// ════════════════════════════════════════════════════════════════
// 3. APLICA OFFSET AO TIMESTAMP UTC
// ════════════════════════════════════════════════════════════════

// ✅ MÉTODO SEGURO: Usa valor absoluto e subtrai/soma conforme sinal
offsetSeconds_ABS := DINT_TO_UDINT(ABS(offsetSeconds));

IF offsetSeconds < 0 THEN
    // Fuso NEGATIVO (Américas): subtrai
    timestampLocal_UDINT := Global.timestampUTC - offsetSeconds_ABS;
ELSE
    // Fuso POSITIVO (Europa, Ásia): soma
    timestampLocal_UDINT := Global.timestampUTC + offsetSeconds_ABS;
END_IF

// ════════════════════════════════════════════════════════════════
// 4. CONVERTE TIMESTAMP PARA DATA/HORA LOCAL
// ════════════════════════════════════════════════════════════════

dtNowLocal := UDINT_TO_DT(timestampLocal_UDINT);
dataNowLocal := TO_DATE(dtNowLocal);

// Extrai hora (0..23)
todNowLocal := DT_TO_TOD(dtNowLocal);
todAsDword := TOD_TO_DWORD(todNowLocal);
hora := DWORD_TO_INT(todAsDword / DWORD#3600000);

// Extrai dia da semana (1=Dom .. 7=Sáb)
diadasemana := UDINT_TO_INT(((timestampLocal_UDINT / 86400) + 4) MOD 7) + 1;

// ════════════════════════════���═══════════════════════════════════
// 5. VERIFICA MUDANÇA DE DATA (Para atualizar cache)
// ════════════════════════════════════════════════════════════════

IF dataNowLocal <> lastCheckedDate THEN
    
    lastCheckedDate := dataNowLocal;
    cachedSpecialDateLimit := -1.0;  // Invalida cache
    
    FOR i := 1 TO Global.NDATASESPECIAIS DO
        
        // ✅ OTIMIZAÇÃO: Early exit se encontrar data vazia
        IF PerVar.DatasEspeciais[i] = DATE#1970-01-01 THEN
            EXIT;  // Resto do array está vazio
        END_IF
        
        // Verifica se é data especial
        IF PerVar.DatasEspeciais[i] = dataNowLocal THEN
            cachedSpecialDateLimit := PerVar.SpecialDaySchedule[i];
            EXIT;  // Encontrou, pára a busca
        END_IF
        
    END_FOR
    
END_IF

// ════════════════════════════════════════════════════════════════
// 6. USA CACHE DE DATA ESPECIAL (Se válido)
// ════════════════════════════════════════════════════════════════

IF cachedSpecialDateLimit >= 0.0 THEN
    // Data especial ativa
    Global.MaxExportLimit := cachedSpecialDateLimit;
    Global.sMessage := 'Agenda: Data especial';
    RETURN;
END_IF

// ════════════════════════════════════════════════════════════════
// 7. AGENDA SEMANAL (Hora Local)
// ════════════════════════════════════════════════════════════════

// ✅ VALIDAÇÃO: Verifica se índices estão dentro dos limites
IF (diadasemana >= 1 AND diadasemana <= 7) AND (hora >= 0 AND hora <= 23) THEN
    
    // Acessa agenda semanal
    Global.MaxExportLimit := PerVar.WeekSchedule_kW[diadasemana, hora + 1];
    Global.sMessage := '';  // ✅ Limpa mensagem de erro anterior
    
ELSE
    
    // ❌ ERRO: Índice inválido (não deveria ocorrer)
    Global.MaxExportLimit := 0.0;
    Global.sMessage := 'ERRO: Índice de agenda inválido';
    Global.K8ErroOut := TRUE;
    
END_IF

END_FUNCTION_BLOCK

// Dispositivo/Application/FB Auxiliares/FB_FFQ
(*
    FB_FFQ - Feedforward de Potência Reativa 
    Função:
    - Calcula o Q MÍNIMO necessário para atingir PF_target
    - Não calcula Q exato, mas o valor mínimo aceitável
    - Se o sistema fornecer menos Q, o PF ficará maior (melhor)
    - Se fornecer mais Q, o PF ficará menor (pior)
    Fórmula:
    Q_min = P × tan(acos(PF_target)) => Simplificado: Q_min = P × √(1 - PF²) / PF
*)

FUNCTION_BLOCK FB_FFQ
VAR_INPUT
    P_active_kW   : REAL;    // Potência ativa comandada (kW)
    PF_target_abs : REAL;    // PF alvo (0.92)
    PF_sign       : REAL;    // 1.0 = indutivo, -1.0 = capacitivo
END_VAR

VAR_OUTPUT
    Q_reactive_kvar : REAL;   // Potência Reativa Calculada (var) - Q mínimo para atingir PF_target
END_VAR

VAR
    tan_phi : REAL;           // Tangente do ângulo de fase
    Q_target    : REAL;       // Q total necessário no ponto de conexão
END_VAR

// 1. Proteção: se potência ativa é zero ou negativa, não há Q a calcular
IF P_active_kW <= 0.0 THEN
    Q_reactive_kvar := 0.0;
    RETURN;
END_IF

// Proteção: PF_target deve estar entre 0 e 1
IF PF_target_abs <= 0.0 OR PF_target_abs > 1.0 THEN
    Q_reactive_kvar := 0.0;
    RETURN;
END_IF

// 2. Q total necessário no ponto de conexão para PF = 0.92
// Método 1: usando tan(acos(PF))
// phi := ACOS(PF_target_abs);              // Ângulo de fase em radianos
// tan_phi := TAN(phi);                     // Tangente do ângulo
// Q_reactive_var := P_active_W * tan_phi;
// Método 2: Simplificado (mais eficiente, evita ACOS e TAN)
// tan(acos(x)) = sqrt(1 - x²) / x
tan_phi := SQRT(1.0 - (PF_target_abs * PF_target_abs)) / PF_target_abs;
Q_target := P_active_kW * tan_phi;

// atribuição correta
Q_reactive_kvar := Q_target;

// 3. Aplica o sinal (Indutivo = positivo, Capacitivo = negativo)
// Nota: Para controle de exportação, normalmente usamos indutivo (Q positivo)
IF PF_sign < 0.0 THEN
    Q_reactive_kvar := -Q_reactive_kvar;  // Capacitivo
END_IF

// Resultado: Q_reactive_var é o Q MÍNIMO para atingir PF_target
// - Se injetar menos Q: PF > PF_target (melhor)
// - Se injetar mais Q: PF < PF_target (pior)
// - Se injetar exatamente Q: PF = PF_target

END_FUNCTION_BLOCK

// Dispositivo/Application/FB Auxiliares/FB_PIQ
(*
    FB_PIQ - Controlador PI para Fator de Potência
    Lógica para PF ≥ 0.92:
    - Se PV (PF medido) ≥ SP (PF target): erro = 0 (objetivo atingido)
    - Se PV < SP: erro = SP - PV (precisa aumentar Q)
    Diferente de um PI normal:
    - Erro ZERO quando PF ≥ target (não tenta melhorar além do necessário)
    - Saída é comando de Q (kvar)
*)

FUNCTION_BLOCK FB_PIQ
VAR_INPUT
    SP : REAL;                      		// Setpoint de PF (0.92)
    PV : REAL;                      		// PF medido (absoluto)
	Kp : REAL;              
    Ki : REAL;              
    CycleTime : REAL;       				
    P_cmd : REAL;                   		// Comando de P (para referência)
    RampUp : REAL;                  		// Rampa de subida (kvar/s)
    RampDown : REAL;                		// Rampa de descida (kvar/s)
    DeadbandAbs : REAL;             		// Zona morta de PF (ex: 0.01)
    Reset : BOOL;                   		// Zera o controlador
    bExternal_Saturated : BOOL := FALSE;  	// NOVO: Saturação externa (de FB_QAlloc)
	OutMax : REAL := 1000.0;    			// Limite superior de MV (kvar)
    OutMin : REAL := 0.0;       			// Limite inferior de MV (kvar)
END_VAR

VAR_OUTPUT
    MV : REAL;                      // Comando de Q (kvar)
    Error : REAL;                   // BOOL → REAL (valor do erro)
    Saturated : BOOL;               // TRUE = saída saturada
END_VAR

VAR
    integral : REAL := 0.0;         // Acumulador integral
    P_term : REAL;                  // Termo proporcional
    I_term : REAL;                  // Termo integral
    MV_raw : REAL;                  // Saída bruta (antes de rampa)
    MV_prev : REAL := 0.0;          // Saída do ciclo anterior
    delta : REAL;                   // Variação desejada
    delta_max : REAL;               // Variação máxima permitida
    erro : REAL;                    // Erro de PF
    sinal_saturacao : INT;      	// para anti-windup direcional
END_VAR

// ════════════════════════════════════════════════════════════════
// 1. RESET
// ════════════════════════════════════════════════════════════════
IF Reset THEN
    integral := 0.0;
    MV := 0.0;
    MV_prev := 0.0;
    Error := 0.0;  
    Saturated := FALSE;
    RETURN;
END_IF

// ════════════════════════════════════════════════════════════════
// 2. CALCULA ERRO COM LÓGICA ESPECIAL (PF ≥ TARGET)
// ════════════════════════════════════════════════════════════════

IF PV >= SP THEN
    erro := 0.0;  // PF medido ≥ PF target: objetivo atingido
ELSE
    erro := SP - PV;  // PF medido < PF target: precisa corrigir
END_IF

Error := erro;  // ✅ Saída do erro

// ════════════════════════════════════════════════════════════════
// 3. ZONA MORTA (DEADBAND)
// ════════════════════════════════════════════════════════════════

IF ABS(erro) < DeadbandAbs THEN
    erro := 0.0;
END_IF

// ════════════════════════════════════════════════════════════════
// 4. CÁLCULO PI
// ════════════════════════════════════════════════════════════════

P_term := Kp * erro;
I_term := integral + (Ki * erro * CycleTime);
MV_raw := P_term + I_term;

// ════════════════════════════════════════════════════════════════
// 5. ✅ SATURAÇÃO COM OutMax/OutMin (ALTERAÇÃO)
// ════════════════════════════════════════════════════════════════
IF MV_raw > OutMax THEN
    MV_raw := OutMax;
    sinal_saturacao := 1;
ELSIF MV_raw < OutMin THEN
    MV_raw := OutMin;
    sinal_saturacao := -1;
ELSE
    sinal_saturacao := 0;
END_IF

// ════════════════════════════════════════════════════════════════
// 6. ANTI-WINDUP (Conditional Integration)
// ════════════════════════════════════════════════════════════════

IF bExternal_Saturated OR (sinal_saturacao <> 0) THEN
    // Saturado: só acumula se erro empurra para FORA da saturação
    IF (sinal_saturacao = 1 AND erro < 0.0) OR
       (sinal_saturacao = -1 AND erro > 0.0) THEN
        integral := I_term;  // Permite desacumular
    END_IF
    // Caso contrário: integral permanece (freeze)
    Saturated := TRUE;
ELSE
    integral := I_term;
    Saturated := FALSE;
END_IF

// ════════════════════════════════════════════════════════════════
// 7. RATE LIMITER (Rampa)
// ════════════════════════════════════════════════════════════════

delta := MV_raw - MV_prev;

IF delta > 0.0 THEN
    delta_max := RampUp * Global.ControlCycle;
    IF delta > delta_max THEN
        MV := MV_prev + delta_max;
    ELSE
        MV := MV_raw;
    END_IF
    
ELSIF delta < 0.0 THEN
    delta_max := RampDown * Global.ControlCycle;
    IF ABS(delta) > delta_max THEN
        MV := MV_prev - delta_max;
    ELSE
        MV := MV_raw;
    END_IF
    
ELSE
    MV := MV_raw;
END_IF

MV_prev := MV;

END_FUNCTION_BLOCK

// Dispositivo/Application/FB Auxiliares/FB_QAlloc

(*
    ════════════════════════════════════════════════════════════════
    FB_QAlloc - Alocador de Potência Reativa
    ════════════════════════════════════════════════════════════════
*)

FUNCTION_BLOCK FB_QAlloc
VAR_INPUT
    Q_total_cmd_kvar : REAL;        // Comando de Q total (do FB_PIQ)
END_VAR

VAR_OUTPUT
    bQ_limit_reached : BOOL;        // TRUE = Não conseguiu alocar todo Q
    Q_allocated_kvar : REAL;        // Q efetivamente alocado
    PF_effective : REAL;            // PF efetivo total resultante
    Q_capacity_total : REAL;        // Capacidade total de Q disponível (kvar)
    S_total_used : REAL;            // S total utilizado (kVA)
END_VAR

VAR

	// ✅ Acumuladores totais
    Q_total : REAL;
    P_total : REAL;
    Q_capacity_total_internal : REAL;
    S_total_used_internal : REAL;

	// ✅ Variáveis por inversor
    Q_target_i : REAL;
    Q_actual_i : REAL;
    Q_max_i : REAL;
    S_available_i : REAL;
    P_actual_i : REAL;
	
    // ✅ Auxiliares
    i : UINT;
    proportion : REAL;
    S_total : REAL;
    S_i : REAL;  // ✅ S do inversor i (calculado 1 vez)
END_VAR

// ════════════════════════════════════════════════════════════════
// INICIALIZAÇÃO
// ════════════════════════════════════════════════════════════════

Q_total := 0.0;
P_total := 0.0;
Q_capacity_total_internal := 0.0;
S_total_used_internal := 0.0;
bQ_limit_reached := FALSE;

// ════════════════════════════════════════════════════════════════
// LOOP PRINCIPAL
// ════════════════════════════════════════════════════════════════

FOR i := 1 TO Global.NMAXINVERSORES DO
    
    IF PerVar.InvActivePower[i] > 0.0 THEN
        
        // ────────────────────────────────────────────────────────
        // A. LÊ P JÁ ALOCADO
        // ────────────────────────────────────────────────────────
        P_actual_i := Global.P_inv_kW[i];
        
        // ────────────────────────────────────────────────────────
        // B. CALCULA Q MÁXIMO DISPONÍVEL
        // ────────────────────────────────────────────────────────
        S_available_i := PerVar.InvSmaxPower[i];
        
        IF S_available_i > ABS(P_actual_i) THEN
            Q_max_i := SQRT((S_available_i * S_available_i) - (P_actual_i * P_actual_i));
        ELSE
            Q_max_i := 0.0;
        END_IF
        
        Global.Inv_Q_available[i] := Q_max_i;
        
        // ─────────────────────────────────────────���──────────────
        // C. DISTRIBUI Q PROPORCIONALMENTE
        // ────────────────────────────────────────────────────────
        IF Global.P_allocated_kW > 0.01 THEN
            proportion := Global.P_inv_kW[i] / Global.P_allocated_kW;
        ELSE
            proportion := 0.0;
        END_IF
        
        Q_target_i := Q_total_cmd_kvar * proportion;
        
        // ────────────────────────────────────────────────────────
        // D. LIMITA Q AO DISPONÍVEL
        // ────────────────────────────────────────────────────────
        IF ABS(Q_target_i) > Q_max_i THEN
            
            IF Q_target_i >= 0.0 THEN
                Q_actual_i := Q_max_i;
            ELSE
                Q_actual_i := -Q_max_i;
            END_IF
            
            bQ_limit_reached := TRUE;
            Global.Inv_limited[i] := TRUE;
            
        ELSE
            Q_actual_i := Q_target_i;
            Global.Inv_limited[i] := FALSE;
        END_IF
        
        // ────────────────────────────────────────────────────────
        // E. ARMAZENA Q
        // ────────────────────���───────────────────────────────────
        Global.Q_inv_kvar[i] := Q_actual_i;
        
        // ────────────────────────────────────────────────────────
        // F. CALCULA S UTILIZADO (✅ UMA VEZ)
        // ────────────────────────────────────────────────────────
        S_i := SQRT((P_actual_i * P_actual_i) + (Q_actual_i * Q_actual_i));
        
        S_total_used_internal := S_total_used_internal + S_i;
        
        // Utilização de S (%)
        IF S_available_i > 0.0 THEN
            Global.Inv_S_utilization[i] := (S_i / S_available_i) * 100.0;
        ELSE
            Global.Inv_S_utilization[i] := 0.0;
        END_IF
        
        // ────────────────────────────────────────────────────────
        // G. CALCULA PF INDIVIDUAL
        // ────────────────────────────────────────────────────────
        IF S_i > 0.01 THEN
            Global.PF_inv[i] := P_actual_i / S_i;
        ELSE
            Global.PF_inv[i] := 1.0;
        END_IF
        
        // ────────────────────────────────────────────────────────
        // H. ACUMULADORES
        // ────────────────────────────────────────────────────────
        P_total := P_total + P_actual_i;
        Q_total := Q_total + Q_actual_i;
        Q_capacity_total_internal := Q_capacity_total_internal + Q_max_i;
        
    ELSE
        // Inversor inativo
        Global.Q_inv_kvar[i] := 0.0;
        Global.PF_inv[i] := 1.0;
        Global.Inv_Q_available[i] := 0.0;
        Global.Inv_S_utilization[i] := 0.0;
        Global.Inv_limited[i] := FALSE;
    END_IF
    
END_FOR

// ════════════════════════════════════════════════════════════════
// SAÍDAS
// ════════════════════════════════════════════════════════════════

Q_allocated_kvar := Q_total;
Q_capacity_total := Q_capacity_total_internal;
S_total_used := S_total_used_internal;

// PF efetivo total
IF P_total > 0.01 OR ABS(Q_total) > 0.01 THEN
    S_total := SQRT((P_total * P_total) + (Q_total * Q_total));
    PF_effective := P_total / S_total;
ELSE
    PF_effective := 1.0;
END_IF

END_FUNCTION_BLOCK

// Dispositivo/Application/FB Auxiliares/FB_PAlloc
(*
    ════════════════════════════════════════════════════════════════
    FB_PAlloc - Alocador de Potência Ativa (PRIORIDADE MÁXIMA)
    ════════════════════════════════════════════════════════════════
*)
FUNCTION_BLOCK FB_PAlloc
VAR_INPUT
    P_total_cmd_kW : REAL;          // Comando de P total (do FB_PI)
END_VAR

VAR_OUTPUT
    P_allocated_kW : REAL;          // ✅ ADICIONAR ESTA SAÍDA!
END_VAR

VAR
    i : UINT;
    P_target_i : REAL;
    P_actual_i : REAL;
    P_total_calc : REAL;
    proportion : REAL;
END_VAR


P_total_calc := 0.0;

FOR i := 1 TO Global.NMAXINVERSORES DO     
    
    IF PerVar.InvActivePower[i] > 0.0 THEN
        
        // Proporção do inversor
        proportion := PerVar.InvActivePower[i] / Global.InstalledPower;
        
        // P proporcional
        P_target_i := P_total_cmd_kW * proportion;
        
        // Limita apenas pela nominal (ignora S_max por enquanto)
        P_actual_i := MIN(P_target_i, PerVar.InvActivePower[i]);
        
        // Armazena P
        Global.P_inv_kW[i] := P_actual_i;
        
        // Setpoint percentual
        IF PerVar.InvActivePower[i] > 0.0 THEN
            Global.P_inv_Percent[i] := (P_actual_i / PerVar.InvActivePower[i]) * 100.0;
        ELSE
            Global.P_inv_Percent[i] := 0.0;
        END_IF
        
        P_total_calc := P_total_calc + P_actual_i;
        
    ELSE
        Global.P_inv_kW[i] := 0.0;
        Global.P_inv_Percent[i] := 0.0;
    END_IF
    
END_FOR

// ✅ ATUALIZA SAÍDA
P_allocated_kW := P_total_calc;

END_FUNCTION_BLOCK

// Dispositivo/Application/FB Auxiliares/FB_PI
FUNCTION_BLOCK FB_PI
VAR_INPUT
    setpoint    : REAL;         		// Setpoint desejado
    feedback    : REAL;         		// Medição atual (feedback)
    Kp          : REAL;         		// Ganho proporcional
    Ki          : REAL;         		// Ganho integral
    OutMax      : REAL;         		// Limite superior de saída
    OutMin      : REAL;         		// Limite inferior de saída
    CycleTime   : REAL;         		// Tempo de ciclo (s)
    RampUp      : REAL := 1.0E+6;  		//  Rampa de subida (unidade/s). Default = sem limite
    RampDown    : REAL := 1.0E+6;  		//  Rampa de descida (unidade/s). Default = sem limite
    Deadband    : REAL := 0.0;          //  deadband em kW (já convertido de %)
    bReset      : BOOL := FALSE;        //  reset do PI
END_VAR

VAR_OUTPUT
    u           : REAL;         		// Saída do controlador
    erro        : REAL;         		// Erro atual (setpoint - feedback)
    bSaturated  : BOOL;         		// TRUE = saída saturada
END_VAR

VAR
    integ           : REAL := 0.0;      // Integral acumulada
    LastOut         : REAL := 0.0;
    erroAtual       : REAL;             // Erro no ciclo atual
    u_prop          : REAL;             // Componente proporcional
    u_raw           : REAL;             // Saída antes da saturação
    u_limited       : REAL;         	// Saída após saturação, antes da rampa
    delta           : REAL;         	// Variação desejada
    delta_max       : REAL;         	// Variação máxima permitida
    primeiro_ciclo  : BOOL := TRUE;     // Flag de primeira execução
    sinal_saturacao : INT;              // +1: saturado max, -1: saturado min, 0: não saturado
END_VAR


// ════════════════════════════════════════════════════════════════
// Reset explícito
// ════════════════════════════════════════════════════════════════
IF bReset THEN
    integ := 0.0;
    LastOut := 0.0;
    u := 0.0;
    bSaturated := FALSE;
    primeiro_ciclo := TRUE;
    RETURN;
END_IF

// ════════════════════════════════════════════════════════════════
// Inicialização suave na primeira execução
// ════════════════════════════════════════════════════════════════
IF primeiro_ciclo THEN
    integ := 0.0;
    primeiro_ciclo := FALSE;
    
    // Se quiser inicializar LastOut com valor atual do medidor:
    // LastOut := feedback;  // Opcional: evita salto inicial
END_IF

// ════════════════════════════════════════════════════════════════
// Cálculo do Erro + Deadband
// ════════════════════════════════════════════════════════════════
erroAtual := setpoint - feedback;

// ✅ Deadband
IF ABS(erroAtual) < Deadband THEN
    erroAtual := 0.0;
END_IF

erro := erroAtual;  // Saída para diagnóstico

// ════════════════════════════════════════════════════════════════
// Componente Proporcional
// ════════════════════════════════════════════════════════════════
u_prop := Kp * erroAtual;

// ════════════════════════════════════════════════════════════════
// Saída Raw (P + I + LastOut)
// ══════════════════════════════════════════���═════════════════════
u_prop := Kp * erroAtual;
u_raw := u_prop + integ;

// ════════════════════════════════════════════════════════════════
// Saturação
// ════════════════════════════════════════════════════════════════
IF u_raw > OutMax THEN
    u_limited := OutMax;
    bSaturated := TRUE;
    sinal_saturacao := 1;
ELSIF u_raw < OutMin THEN
    u_limited := OutMin;
    bSaturated := TRUE;
    sinal_saturacao := -1;
ELSE
    u_limited := u_raw;
    bSaturated := FALSE;
    sinal_saturacao := 0;
END_IF

// ════════════════════════════════════════���═══════════════════════
// Rate Limiter (Rampa)
// ════════════════════════════════════════════════════════════════
delta := u_limited - LastOut;

IF delta > 0.0 THEN
    delta_max := RampUp * CycleTime;
    IF delta > delta_max THEN
        u := LastOut + delta_max;
    ELSE
        u := u_limited;
    END_IF
ELSIF delta < 0.0 THEN
    delta_max := RampDown * CycleTime;
    IF ABS(delta) > delta_max THEN
        u := LastOut - delta_max;
    ELSE
        u := u_limited;
    END_IF
ELSE
    u := u_limited;
END_IF
// ════════════════════════════════════════════════════════════════
// Anti-windup Melhorado (Conditional Integration)
// ════════════════════════════════════════════════════════════════
// Regras:
// 1. NÃO saturado → acumula normalmente
// 2. Saturado MAS erro na direção oposta → permite desacumular
// 3. Saturado E erro na mesma direção → freeze (não acumula)

IF NOT bSaturated THEN
    // Caso 1: Normal - acumula integral
    integ := integ + (Ki * erroAtual * CycleTime);
    
ELSIF (sinal_saturacao = 1 AND erroAtual < 0.0) OR (sinal_saturacao = -1 AND erroAtual > 0.0) THEN
    // Caso 2: Saturado MAS erro está tentando sair da saturação
    // Permite acumular para ajudar a desaturar
    integ := integ + (Ki * erroAtual * CycleTime);
    
ELSE
    // Caso 3: Saturado E erro empurrando mais para saturação
    // NÃO acumula (freeze integral)
    // integ permanece inalterado
END_IF

// ════════════════════════════════════════════════════════════════
// Atualiza LastOut
// ════════════════════════════════════════════════════════════════
LastOut := u;

END_FUNCTION_BLOCK

// Dispositivo/Application/FB Auxiliares/FB_Diagnostico
(*
    ════════════════════════════════════════════════════════════════
    FB_Diagnostico - Diagnóstico de Fator de Potência
    ════════════════════════════════════════════════════════════════
    
    Gera diagnóstico completo do sistema de compensação de PF,
    incluindo alarmes, recomendações e estatísticas.
    
    ═══���════════════════════════════════════════════════════════════
*)

FUNCTION_BLOCK FB_Diagnostico
VAR_INPUT
    P_allocated_kW : REAL;
    Q_commanded_kvar : REAL;
    Q_allocated_kvar : REAL;
    Q_capacity_kvar : REAL;
    PF_measured : REAL;
    PF_achieved : REAL;
    bQ_limited : BOOL;
END_VAR

VAR
    Q_deficit : REAL;
    Q_deficit_pct : REAL;
    S_total_avail : REAL;
    S_total_used : REAL;
    bank_size : REAL;
    bank_size_int : DINT;  // ✅ DINT (não INT)
END_VAR

// ════════════════════════════════════════════════════════════════
// 1. ARMAZENA VALORES BÁSICOS
// ════════════════════════════════════════════════════════════════

Global.P_generated_kW := P_allocated_kW;
Global.P_allocated_kW := P_allocated_kW;
Global.Q_commanded_kvar := Q_commanded_kvar;
Global.Q_allocated_kvar := Q_allocated_kvar;
Global.Q_available_kvar := Q_capacity_kvar;
Global.PF_measured := PF_measured;
Global.PF_achieved := PF_achieved;

// Q medido (do ponto de conexão)
Global.Q_measured_kvar := Global.Qt;  // Já convertido em kvar pelo FB_AjustaLeitura

// ════════════════════════════════════════════════════════════════
// 2. CALCULA DÉFICIT DE Q
// ════════════════════════════════════════════════════════════════

Q_deficit := Q_commanded_kvar - Q_allocated_kvar;
Global.Q_deficit_kvar := Q_deficit;

// Déficit percentual
IF ABS(Q_commanded_kvar) > 0.1 THEN
    Q_deficit_pct := (ABS(Q_deficit) / ABS(Q_commanded_kvar)) * 100.0;
ELSE
    Q_deficit_pct := 0.0;
END_IF
Global.Q_deficit_percent := Q_deficit_pct;

// ════════════════════════════════════════════════════════════════
// 3. CALCULA UTILIZAÇÃO DE S
// ════════════════════════════════════════════════════════════════

// S total disponível
S_total_avail := Global.InstalledSmax;
Global.S_total_available_kVA := S_total_avail;

// S total usado
S_total_used := SQRT((P_allocated_kW * P_allocated_kW) + (Q_allocated_kvar * Q_allocated_kvar));
Global.S_total_used_kVA := S_total_used;

// Utilização percentual
IF S_total_avail > 0.0 THEN
    Global.S_utilization_pct := (S_total_used / S_total_avail) * 100.0;
ELSE
    Global.S_utilization_pct := 0.0;
END_IF

// ════════════════════════════════════════════════════════════════
// 4. CALCULA UTILIZAÇÃO DE Q
// ════════════════════════════════════════════════════════════════

Global.Q_capacity_total_kvar := Q_capacity_kvar;

IF Q_capacity_kvar > 0.0 THEN
    Global.Q_utilization_pct := (ABS(Q_allocated_kvar) / Q_capacity_kvar) * 100.0;
ELSE
    Global.Q_utilization_pct := 0.0;
END_IF

// ════════════════════════════════════════════════════════════════
// 5. CALCULA TAMANHO DE BANCO DE CAPACITORES
// ════════════════════════════════════════════════════════════════

IF Q_deficit > 0.1 THEN
    // Adiciona 10% de margem
    bank_size := ABS(Q_deficit) * 1.1;
	bank_size := DINT_TO_REAL(TRUNC(bank_size / 5.0) + 1) * 5.0;
    Global.Capacitor_bank_size_kvar := bank_size;
    Global.Capacitor_bank_recommended := TRUE;
ELSE
    Global.Capacitor_bank_size_kvar := 0.0;
    Global.Capacitor_bank_recommended := FALSE;
END_IF

// ════════════════════════════════════════════════════════════════
// 6. DETERMINA STATUS DE PF
// ════════════════════════════════════════════════════════════════

IF PF_achieved >= Global.PF_target THEN
    Global.PF_OK := TRUE;
    Global.PFErro := FALSE;
    Global.PF_alarm_code := 0;  // OK
    Global.PF_alarm_message := 'Fator de Potencia OK';
ELSE
    Global.PF_OK := FALSE;
    
    IF bQ_limited THEN
        Global.PFErro := TRUE;
        
        // Classifica severidade
        IF Q_deficit_pct > 20.0 THEN
            Global.PF_alarm_code := 2;  // Crítico
            Global.PF_alarm_message := 'CRITICO: Limite de Q atingido - Banco de capacitores necessario';
        ELSE
            Global.PF_alarm_code := 1;  // Aviso
            Global.PF_alarm_message := 'AVISO: Limite de Q atingido - Considerar banco de capacitores';
        END_IF
    ELSE
        // PF < 0.92 mas não por limite de Q (transitório)
        Global.PFErro := FALSE;
        Global.PF_alarm_code := 1;
        Global.PF_alarm_message := 'PF abaixo do alvo - Sistema compensando';
    END_IF
END_IF

// ════════════════════════════════════════════════════════════════
// 7. ATUALIZA HISTÓRICO (OPCIONAL - implementar com timers)
// ════════════════════════════════════════════════════════════════

// Atualiza PF mínimo
IF PF_achieved < Global.PF_min_24h THEN
    Global.PF_min_24h := PF_achieved;
END_IF

// Atualiza déficit máximo
IF Q_deficit > Global.Q_deficit_max_24h THEN
    Global.Q_deficit_max_24h := Q_deficit;
END_IF

// Conta alarmes (incrementar quando alarme dispara pela primeira vez)
// (Implementar com edge detection)

END_FUNCTION_BLOCK

// Dispositivo/Application/FB Auxiliares/FB_PowerController
(*
    ════════════════════════════════════════════════════════════════
    FB_PowerController - Controlador de Potência Ativa
    ════════════════════════════════════════════════════════════════
    
    Responsabilidade:
    - Calcular comando de P (PI + Safety Margin + Limites de Fase)
    - Encapsular toda lógica relacionada a potência ativa
    
    Pipeline:
    1. PI → P_cmd_raw
    2. Safety Margin → P_cmd_with_margin
    3. Limitador de Fase → P_cmd_limited
    
    ════════════════════════════════════════════════════════════════
*)
FUNCTION_BLOCK FB_PowerController
VAR_INPUT
    ExportLimit_kW : REAL;      // Do scheduler (kW)
    Feedback_kW : REAL;         // Leitura do medidor (kW)
    bReset : BOOL;              // Reset do PI
END_VAR

VAR_OUTPUT
    P_cmd_kW : REAL;            // Comando final (kW)
    bSaturated : BOOL;          // PI saturado
    bPhase_limited : BOOL;      // Limitado por fase
    sLimited_phase : STRING;    // Qual fase limitou
    Margin_applied_kW : REAL;   // Margem aplicada (telemetria)
	EffectiveExportLimit_kW : REAL;
END_VAR

VAR
    // Sub-blocos
    fbPI : FB_PI;
    fbSafetyMargin : FB_SafetyMargin;
    fbFLimiter : FB_FLimiter;
	fbDroop : FB_DroopP;
    
    // Variáveis internas
    P_setpoint : REAL;
    P_cmd_raw : REAL;
    P_cmd_with_margin : REAL;
	lastInstalledPower : REAL := -1.0;
	
	// Droop
    P_error_kW : REAL;
    P_droop_kW : REAL;
	
    P_droop_max_kW : REAL;
    P_cmd_sum : REAL;
	
	// ✅ Deadband em kW (convertido de %)
	Deadband_P_kW     : REAL;
    Droop_Deadband_kW : REAL;
END_VAR

// ────────────────────────────────────────────────────────────────
// ETAPA 1: CONTROLADOR PI
// ────────────────────────────────────────────────────────────────

// Setpoint negativo (exportação)
P_setpoint := -ABS(ExportLimit_kW);

// Erro (kW)
P_error_kW := Feedback_kW - P_setpoint;

// Converte deadband (%) para kW (mínimo 1 kW)
// Recalcula apenas se InstalledPower mudou
IF lastInstalledPower <> Global.InstalledPower THEN
    Deadband_P_kW := MAX(1.0, Global.InstalledPower * (PerVar.Deadband_P / 100.0));
    Droop_Deadband_kW := MAX(1.0, Global.InstalledPower * (PerVar.Deadband_Droop / 100.0));
	Deadband_P_kW := MIN(20.0, MAX(1.0, Global.InstalledPower * (PerVar.Deadband_P / 100.0)));
	Droop_Deadband_kW := MIN(20.0, MAX(1.0, Global.InstalledPower * (PerVar.Deadband_Droop / 100.0)));		
    lastInstalledPower := Global.InstalledPower;
END_IF

// Limite máximo do droop (fração da potência instalada)
P_droop_max_kW := PerVar.Droop_Max * Global.InstalledPower;

// Calcula droop
fbDroop(
    Enable      := PerVar.Droop_Enable,
    bReset      := bReset,                 
    Error_kW    := P_error_kW,
    K_droop     := PerVar.K_Droop,
    Deadband_kW := Droop_Deadband_kW,
    P_max_kW    := P_droop_max_kW
);

P_droop_kW := fbDroop.P_droop_kW;

// PI de potência ativa
fbPI(
    setpoint    := P_error_kW,
    feedback    := 0.0,
    Kp          := PerVar.Kp_P,
    Ki          := PerVar.Ki_P,
    OutMax      := Global.InstalledPower,
    OutMin      := 0.0,
    CycleTime   := Global.ControlCycle,
	RampUp      := PerVar.RampUp_P,     
    RampDown    := PerVar.RampDown_P,    
    Deadband    := Deadband_P_kW,
	bReset      := bReset          
);

// Soma droop + PI
P_cmd_sum := P_droop_kW + fbPI.u;

// Comando bruto (segue fluxo normal)
P_cmd_raw := P_cmd_sum;
IF P_cmd_raw < 0.0 THEN
    P_cmd_raw := 0.0;
ELSIF P_cmd_raw > Global.InstalledPower THEN
    P_cmd_raw := Global.InstalledPower;
END_IF
bSaturated := fbPI.bSaturated;

// ─────────────────────────────────────────���──────────────────────
// ETAPA 2: SAFETY MARGIN
// ────────────────────────────────────────────────────────────────

fbSafetyMargin(
    P_cmd_raw_kW := P_cmd_raw,
    Margin_pct := PerVar.SafetyMargin_pct,
    TC_Power_kW := PerVar.TC_Power_kW
);

P_cmd_with_margin := fbSafetyMargin.P_cmd_adjusted_kW;
Margin_applied_kW := fbSafetyMargin.Margin_applied_kW;  // ✅ Telemetria
EffectiveExportLimit_kW := P_setpoint + Margin_applied_kW;
// ────────────────────────────────────────────────────────────────
// ETAPA 3: LIMITADOR DE FASE
// ────────────────────────────────────────────────────────────────

fbFLimiter(
    P_cmd_in := P_cmd_with_margin,
    PowerMode := PerVar.PowerMode
);

P_cmd_kW := fbFLimiter.P_cmd_out;
bPhase_limited := fbFLimiter.bPhase_limited;
sLimited_phase := fbFLimiter.sLimited_phase;

// ────────────────────────────────────────────────────────────────
// PROTEÇÃO FINAL: Potência Instalada
// ────────────────────────────────────────────────────────────────

IF P_cmd_kW > Global.InstalledPower THEN
    P_cmd_kW := Global.InstalledPower;
    bSaturated := TRUE;
END_IF

END_FUNCTION_BLOCK

// Dispositivo/Application/FB Auxiliares/FB_SafetyMargin
(*
    ════════════════════════════════════════════════════════════════
    FB_SafetyMargin - Margem de Segurança para Correção de TC
    ════════════════════════════════════════════════════════════════
    
    Função:
    - Aplica margem de segurança para compensar erro de TC em baixas correntes
    - Desloca setpoint para lado da importação (garante não exportar)
    
    Exemplo:
    - P_cmd = 100 kW
    - TC_Power = 329 kW
    - Margin = 3%
    - SafetyMargin = 3% × 329 = 9.87 kW
    - P_adjusted = 100 - 9.87 = 90.13 kW
    ════════════════════════════════════════════════════════════════
*)
FUNCTION_BLOCK FB_SafetyMargin
VAR_INPUT
    P_cmd_raw_kW : REAL;        // Comando sem margem
    Margin_pct : REAL;          // Percentual (ex: 3.0)
    TC_Power_kW : REAL;         // Potência do TC
END_VAR

VAR_OUTPUT
    P_cmd_adjusted_kW : REAL;   // Comando com margem
    Margin_applied_kW : REAL;   // Margem aplicada (para telemetria)
END_VAR

VAR
    SafetyMargin_kW : REAL;
END_VAR

// ════════════════════════════════════════════════════════════════
// IMPLEMENTAÇÃO
// ════════════════════════════════════════════════════════════════
// 1. Proteção: se TC não configurado, não aplica margem
IF TC_Power_kW <= 0.0 THEN
    P_cmd_adjusted_kW := P_cmd_raw_kW;
    Margin_applied_kW := 0.0;
    RETURN;
END_IF

// 2. Calcula margem em kW
SafetyMargin_kW := (Margin_pct / 100.0) * TC_Power_kW;

// 3. Aplica margem (reduz comando)
P_cmd_adjusted_kW := P_cmd_raw_kW - SafetyMargin_kW;

// 4. Limita para não ficar negativo
IF P_cmd_adjusted_kW < 0.0 THEN
    P_cmd_adjusted_kW := 0.0;
END_IF

// 5. Armazena margem aplicada (para HMI)
Margin_applied_kW := SafetyMargin_kW;

END_FUNCTION_BLOCK

// Dispositivo/Application/FB Auxiliares/FB_FLimiter
(*
    FB_FLimiter - Limitador por Fase
    
    Função:
    - Verifica se o comando causaria EXPORTAÇÃO excessiva em alguma fase
    - Se fase está IMPORTANDO: ignora (não há problema)
    - Se fase está EXPORTANDO: verifica se comando excederia limite
    
    Lógica:
    1. Calcula P futuro por fase = P_atual + (P_cmd / 3)
    2. Para cada fase EXPORTANDO (P < 0):
       - Verifica se P_futuro < P_phase_limit (mais exportação que permitido)
       - Se sim, calcula comando máximo para essa fase
    3. Usa o MENOR comando máximo entre as fases
    
    Convenção de sinais:
    - P > 0: Importação
    - P < 0: Exportação
    - MaxExportLimit: VALOR POSITIVO na agenda (ex: 90 kW)
    - P_phase_limit: NEGATIVO internamente (ex: -30 kW)
	    
    Exemplo:
    - Agenda: MaxExportLimit = 90 kW (sem sinal)
    - Internamente: P_phase_limit = -90/3 = -30 kW por fase
    - Se Pa = -25 kW (exportando 25 kW)
    - Se P_cmd = -18 kW (quer aumentar exportação)
    - P_future_A = -25 + (-18/3) = -31 kW → EXCEDE -30 kW → LIMITA
*)

FUNCTION_BLOCK FB_FLimiter
VAR_INPUT
    P_cmd_in : REAL;                // Comando de P calculado pelo PI (kW)
    PowerMode : UINT;               // 0=Total, 1=Por fase, 2=Ambos
END_VAR

VAR_OUTPUT
    P_cmd_out : REAL;               // Comando de P limitado por fase (kW)
    bPhase_limited : BOOL;          // TRUE = alguma fase limitou
	sLimited_phase : STRING;        // Qual fase limitou: 'A', 'B', 'C', 'AB', etc.
END_VAR

VAR
    P_cmd_per_phase : REAL;         // Comando adicional por fase (kW)
    P_future_A : REAL;              // P futuro na fase A após aplicar comando (kW)
    P_future_B : REAL;              // P futuro na fase B após aplicar comando (kW)
    P_future_C : REAL;              // P futuro na fase C após aplicar comando (kW)
    P_phase_limit : REAL;           // Limite de exportação por fase (kW negativo)
    P_max_cmd_A : REAL;             // Comando máximo permitido para fase A (kW)
    P_max_cmd_B : REAL;             // Comando máximo permitido para fase B (kW)
    P_max_cmd_C : REAL;             // Comando máximo permitido para fase C (kW)
    P_max_cmd_total : REAL;         // Comando máximo total permitido (kW)
	NO_LIMIT : REAL;                // Constante para "sem limite"
    bLimitA : BOOL;                 // Fase A está limitando
    bLimitB : BOOL;                 // Fase B está limitando
    bLimitC : BOOL;                 // Fase C está limitando
END_VAR

// Comando adicional por fase (distribuído equilibradamente)
P_cmd_per_phase := P_cmd_in / 3.0;

// Limite de exportação por fase
// Se MaxExportLimit = -90 kW, então por fase = -30 kW
P_phase_limit := -ABS(Global.MaxExportLimit) / 3.0;

// ════════════════════════════════════════════════════════════════
// ════════════════════════════════════════════════════════════════
// Inicialização
// ════════════════════════════════════════════════════════════════
NO_LIMIT := Global.InstalledPower * 10.0;  // Valor grande, mas realista
sLimited_phase := '';
bLimitA := FALSE;
bLimitB := FALSE;
bLimitC := FALSE;

// ════════════════════════════════════════════════════════════════
// Se PowerMode = 0, não verifica fase
// ════════════════════════════════════════════════════════════════
IF PowerMode = 0 THEN
    P_cmd_out := P_cmd_in;
    bPhase_limited := FALSE;
    RETURN;
END_IF

// ════════════════════════════════════════════════════════════════
// Proteção: Se InstalledPower não configurado
// ════════════════════════════════════════════════════════════════
IF Global.InstalledPower <= 0.0 THEN
    P_cmd_out := 0.0;
    bPhase_limited := TRUE;
    sLimited_phase := 'ERROR: InstalledPower=0';
    RETURN;
END_IF

// ════════════════════════════════════════════════════════════════
// Calcula P futuro em cada fase após aplicar comando
// ════════════════════════════════════════════════════════════════
P_future_A := Global.Pa + P_cmd_per_phase;
P_future_B := Global.Pb + P_cmd_per_phase;
P_future_C := Global.Pc + P_cmd_per_phase;

// ════════════════════════════════════════════════════════════════
// Verifica FASE A
// ════════════════════════════════════════════════════════════════
IF P_future_A < 0.0 THEN
    // Fase A estará EXPORTANDO após aplicar comando
    
    IF P_future_A < P_phase_limit THEN
        // Excederia o limite de exportação!
        // Calcula quanto PODE aumentar exportação sem exceder:
        // P_max_per_phase = P_limit - P_atual
        // P_max_total = P_max_per_phase * 3
        P_max_cmd_A := (P_phase_limit - Global.Pa) * 3.0;
        bLimitA := TRUE;
    ELSE
        // Dentro do limite: sem restrição
        P_max_cmd_A := NO_LIMIT;
    END_IF
    
ELSE
    // Fase A estará IMPORTANDO: sem problema
    P_max_cmd_A := NO_LIMIT;
END_IF

// ════════════════════════════════════════════════════════════════
// Verifica FASE B
// ════════════════════════════════════════════════════════════════
IF P_future_B < 0.0 THEN
    // Fase B estará EXPORTANDO
    
    IF P_future_B < P_phase_limit THEN
        P_max_cmd_B := (P_phase_limit - Global.Pb) * 3.0;
        bLimitB := TRUE;
    ELSE
        P_max_cmd_B := NO_LIMIT;
    END_IF
    
ELSE
    // Fase B estará IMPORTANDO
    P_max_cmd_B := NO_LIMIT;
END_IF

// ════════════════════════════════════════════════════════════════
// Verifica FASE C
// ════════════════════════════════════════════════════════════════
IF P_future_C < 0.0 THEN
    // Fase C estará EXPORTANDO
    
    IF P_future_C < P_phase_limit THEN
        P_max_cmd_C := (P_phase_limit - Global.Pc) * 3.0;
        bLimitC := TRUE;
    ELSE
        P_max_cmd_C := NO_LIMIT;
    END_IF
    
ELSE
    // Fase C estará IMPORTANDO
    P_max_cmd_C := NO_LIMIT;
END_IF

// ════════════════════════════════════════════════════════════════
// Aplica o MENOR limite (fase mais restritiva)
// ════════════════════════════════════════════════════════════════
P_max_cmd_total := MIN(P_max_cmd_A, MIN(P_max_cmd_B, P_max_cmd_C));

// ════════════════════════════════════════════════════════════════
// Verifica se houve limitação
// ════════════════════════════════════════════════════════════════
IF P_cmd_in > P_max_cmd_total THEN
    P_cmd_out := P_max_cmd_total;
    bPhase_limited := TRUE;
    
    // Identifica qual(is) fase(s) limitou
    IF bLimitA THEN sLimited_phase := CONCAT(sLimited_phase, 'A'); END_IF
    IF bLimitB THEN sLimited_phase := CONCAT(sLimited_phase, 'B'); END_IF
    IF bLimitC THEN sLimited_phase := CONCAT(sLimited_phase, 'C'); END_IF
    
ELSE
    P_cmd_out := P_cmd_in;
    bPhase_limited := FALSE;
    sLimited_phase := '';
END_IF

END_FUNCTION_BLOCK

// Dispositivo/Application/FB Auxiliares/FB_DroopP
(*
    FB_DroopP - Droop para Potência Ativa
    Gera um comando base proporcional ao erro de potência.
    Uso: antes do PI (PI corrige residual).
*)
FUNCTION_BLOCK FB_DroopP
VAR_INPUT
    Enable        : BOOL;   // Habilita droop
    bReset        : BOOL;   // Reset do droop
    Error_kW      : REAL;   // Erro (Setpoint - Feedback)
    K_droop       : REAL;   // Ganho droop (kW/kW)
    Deadband_kW   : REAL;   // Zona morta
    P_max_kW      : REAL;   // Limite absoluto do droop (kW)
END_VAR

VAR_OUTPUT
    P_droop_kW    : REAL;   // Saída do droop (kW)
END_VAR

VAR
    P_cmd : REAL;
    erro  : REAL;
END_VAR

// ──────────────────────────────────��───────────────────────────
// Reset
// ──────────────────────────────────────────────────────────────
IF bReset THEN
    P_droop_kW := 0.0;
    RETURN;
END_IF

// ──────────────────────────────────────────────────────────────
// Lógica do droop
// ──────────────────────────────────────────────────────────────
IF NOT Enable THEN
    P_droop_kW := 0.0;
    RETURN;
END_IF

// Aplica deadband ao erro
erro := Error_kW;
IF ABS(erro) < Deadband_kW THEN
    erro := 0.0;
END_IF

P_cmd := K_droop * erro;

// Limite absoluto
IF P_cmd > P_max_kW THEN
    P_cmd := P_max_kW;
ELSIF P_cmd < -P_max_kW THEN
    P_cmd := -P_max_kW;
END_IF

P_droop_kW := P_cmd;

END_FUNCTION_BLOCK

// Dispositivo/Application/FB_Alarmes
FUNCTION_BLOCK FB_Alarmes
VAR_INPUT
	codigo			: UDINT;
	tError			: UDINT;
END_VAR


CASE codigo OF
	
	// mensagens do driver modbus
	16#0 : Global.sMessage:= 'Sucesso';
	16#1 : Global.sMessage:= 'Código de função não aceito';
	16#2 : Global.sMessage:= 'Deslocamento de registro não permitido';
	16#3 : Global.sMessage:= 'Valor a ser gravado é inválido';
	16#4 : Global.sMessage:= 'Erro irrecuperável ao executar a solicitação';
	16#5 : Global.sMessage:= 'Notificação de um dispositivo escravo de que uma operação demorada foi iniciada';
	16#6 : Global.sMessage:= 'Notificação de um dispositivo escravo de que uma operação demorada está em andamento';
	16#8 : Global.sMessage:= 'Erro específico para os códigos de função 20 e 21';
	16#A : Global.sMessage:= 'Erro específico ao usar dispositivos atrás de um gateway';
	16#B : Global.sMessage:= 'Erro específico ao usar dispositivos atrás de um gateway';
	16#A1: Global.sMessage:= 'Não houve resposta a tempo';
	16#A2: Global.sMessage:= 'O checksum da resposta está incorreto';
	16#A3: Global.sMessage:= 'A resposta não é do dispositivo escravo esperado';
	16#A4: Global.sMessage:= 'A resposta não corresponde ao código de função esperado';
	16#A5: Global.sMessage:= 'Erro na porta TCP. A solicitação não foi enviada';
	16#A6: Global.sMessage:= 'A resposta contém dados inválidos';
	16#A7: Global.sMessage:= 'A resposta não está no protocolo Modbus';
	16#A8: Global.sMessage:= 'Algum campo do cabeçalho Modbus MBAP (Protocolo, Comprimento) é inválido';
	16#A9: Global.sMessage:= 'Algum parâmetro de entrada da operação é inválido';
	16#FF: Global.sMessage:= 'O resultado da solicitação é indefinido ou ainda desconhecido';
	
	// mensagens da aplicação
	16#B1: Global.sMessage:= 'Comunicação modbus foi abortada';
	16#B2: Global.sMessage:= 'Timeout na comunicação modbus';
	

END_CASE

END_FUNCTION_BLOCK

// Dispositivo/Application/FB_ReadMedidor
FUNCTION_BLOCK FB_ReadMedidor

VAR_INPUT
    Execute 				: BOOL;                 // habilita leitura
END_VAR

VAR_OUTPUT
    result 					: E_ModbusResult;      		 // resultado
    bDadosOK				: BOOL:= FALSE;  // Dados aprovados
	bPoucosErros			: BOOL:= TRUE;  // Inicialmente sem erros
END_VAR

VAR
	fbAlarmes				: FB_Alarmes;		 		// converte códigos de erros em mensagens texto
	fbChannel       		: ModbusChannel;
	fbValidaDadosRele		: FB_ValidaDadosRele;	
	
    state 					: (TRIG, WAIT) := TRIG;
	tonTimer				: TON;
	tTimeout				: TIME := T#250MS;			// tempo de leitura do medidor é cerca de 200 ms
END_VAR

// ============================================================
// Máquina de estados de leitura do medidor
// ============================================================

// estado default por ciclo
result := E_ModbusResult.BUSY;

// se não habilitado, não executa
IF NOT Execute THEN
    result := E_ModbusResult.END;
    Global.trigMedidor100 := FALSE;
	state := TRIG;
    RETURN;
END_IF

tonTimer(IN := (state = WAIT), PT := tTimeout);

CASE state OF

    TRIG:
        Global.trigMedidor100 := TRUE;      // trigger rising edge
        state := WAIT;

    WAIT:
        IF Global.pMedidor100^.xDone THEN
            Global.trigMedidor100 := FALSE;
            state := TRIG;
          	result := E_ModbusResult.DONE;
			fbValidaDadosRele();
			bDadosOK:=fbValidaDadosRele.bDadosOK;
			bPoucosErros:=fbValidaDadosRele.bPoucosErros;
			
        ELSIF Global.pMedidor100^.xError THEN
				fbChannel(Slave := Global.pMedidor100^,iChannelIndex := 0);
				fbAlarmes(codigo := fbChannel.ModbusError,tError:=TO_UDINT(SysTimeRtcGet(Global.Result)));
				state:= TRIG;
				Global.trigMedidor100:=FALSE;
          		result := E_ModbusResult.ERRO;
				
		ELSIF tonTimer.Q THEN
				fbAlarmes(codigo := 16#B2,tError:=TO_UDINT(SysTimeRtcGet(Global.Result)));
				state:= TRIG;
				Global.trigMedidor100:=FALSE;	
				result := E_ModbusResult.TIMEOUT;
		END_IF	

END_CASE

END_FUNCTION_BLOCK

// Dispositivo/Application/FB_ValidaDadosRele
(*═════════════════════════════════════════════════════════════════════
 FB_ValidaMedicao
 
 Valida medições do medidor trifásico via Modbus, aplica filtro
 passa-baixa e verifica consistência física das grandezas.
 
 ENTRADAS:
 - (nenhuma - lê de valorLido.WordArray via Modbus)
 
 SAÍDAS:
 - bDadosOK: TRUE se medições são válidas
 - bPoucosErros: TRUE se < 5 erros consecutivos
 - diagnosticCode: Código de falha (0 = OK)
 
 LÓGICA:
 1. Conversão de escalas (Modbus → unidades físicas)
 2. Validação de ranges individuais
 3. Validação cruzada (Pt vs soma, PF vs P/S)
 4. Detecção de congelamento 
 5. Filtro passa-baixa exponencial (SOMENTE se validação OK)
 6. Atualização de variáveis globais (SOMENTE se validação OK)
 7. Janela de erros (5 consecutivos = FAIL_SAFE)
═════════════════════════════════════════════════════════════════════*)
FUNCTION_BLOCK FB_ValidaDadosRele

VAR_OUTPUT
    bDadosOK		: BOOL 	:= FALSE;  // Dados aprovados
	bPoucosErros	: BOOL  := TRUE;  // Inicialmente sem erros
    diagnosticCode 	: WORD;            // Código de falha
END_VAR

VAR
	valorLido		: UN_Rele;
	Ua    	    	: REAL := 0.0; // 2006H - Tensão de fase A x 0,1 V
	Ub    	    	: REAL := 0.0; // 2008H - Tensão de fase B x 0,1 V
	Uc    	    	: REAL := 0.0; // 200AH - Tensão de fase C x 0,1 V
	
	Ia    	    	: REAL := 0.0; // 200CH - Corrente de fase A x 0,001 A 
	Ib    	    	: REAL := 0.0; // 200EH - Corrente de fase B x 0,001 A
	Ic    	    	: REAL := 0.0; // 2010H - Corrente de fase C x 0,001 A
	
	Pt    	    	: REAL := 0.0; // 2012H - Potencia ativa combinada x 0,1 W
	Pa    	    	: REAL := 0.0; // 2014H - Potencia ativa fase A x 0,1 W
	Pb    	    	: REAL := 0.0; // 2016H - Potencia ativa fase B x 0,1 W
	Pc    	   		: REAL := 0.0; // 2018H - Potencia ativa fase C x 0,1 W	
		
	Qt    	    	: REAL := 0.0; // 201AH - Potencia reativa combinada x 0,1 var
	Qa    	    	: REAL := 0.0; // 201CH - Potencia reativa fase A x 0,1 var
	Qb    	    	: REAL := 0.0; // 201EH - Potencia reativa fase B x 0,1 var
	Qc    	    	: REAL := 0.0; // 2020H - Potencia reativa fase C x 0,1 var

	PFt    	    	: REAL := 0.0; // 202AH - Fator de potência combinado (número positivo: indutivo, número negativo: capacitivo) (x  0,001)
	PFa    	    	: REAL := 0.0; // 202CH - Fator de potência de fase A (número positivo: indutivo, número negativo: capacitivo)  (×0,001)
	PFb    	    	: REAL := 0.0; // 202EH - Fator de potência de fase B (número positivo: indutivo, número negativo: capacitivo)  (×0,001)
	PFc    	    	: REAL := 0.0; // 2030H - Fator de potência de fase C (número positivo: indutivo, número negativo: capacitivo)  (×0,001)
	
	// Limites físicos (ajustar conforme instalação)
    PFMIN 			: REAL := 0.5;
    PFMAX 			: REAL := 1.0;
	
	// variaveis auxiliares
    bRangeError 	: BOOL := FALSE;            // Fora de faixa
	nErrors 		: UINT := 0;
	SomaP			: REAL;
	SomaQ 			: REAL;
	Calculado 		: REAL;
	Tolerancia  	: REAL :=0.05;
	Pt_last 		: REAL := 0.0;
    frozen_count 	: UINT := 0;
	FREEZE_THRESHOLD: UINT := 10;  		// 10 ciclos
	bFirstRun		: BOOL :=TRUE;
	Pt_filt 		: REAL :=0;
    Qt_filt 		: REAL :=0;
    PFt_filt 		: REAL :=0;
END_VAR

// ═══════════════════════════════════════════════════════════════
// 1. RESET DE ESTADO
// ═══════════════════════════════════════════════════════════════

bRangeError := FALSE;
diagnosticCode := 0;

// ═══════════════════════════════════════════════════════════════
// 2. CONVERSÃO DE ESCALAS
// ═══════════════════════════════════════════════════════════════
Ua  := valorLido.EmReal.Ua * 0.1;				// em Volts
Ub  := valorLido.EmReal.Ub * 0.1;				// em Volts
Uc  := valorLido.EmReal.Uc * 0.1;				// em Volts

Ia  := valorLido.EmReal.Ia * 0.001;				// em Amperes
Ib  := valorLido.EmReal.Ib * 0.001;				// em Amperes
Ic  := valorLido.EmReal.Ic * 0.001;				// em Amperes

Pt  := valorLido.EmReal.Pt *0.0001;				// kW
Pa  := valorLido.EmReal.Pa *0.0001;				// kW
Pb  := valorLido.EmReal.Pb *0.0001;				// kW
Pc  := valorLido.EmReal.Pc *0.0001;				// kW

Qt  := valorLido.EmReal.Qt *0.0001;				// kvar
Qa  := valorLido.EmReal.Qa *0.0001;				// kvar
Qb  := valorLido.EmReal.Qb *0.0001;				// kvar
Qc  := valorLido.EmReal.Qc *0.0001;				// xkvar

PFt := valorLido.EmReal.PFt *0.001;	
PFa := valorLido.EmReal.PFa *0.001;
PFb := valorLido.EmReal.PFb *0.001;
PFc := valorLido.EmReal.PFc *0.001;

// ═══════════════════════════════════════════════════════════════
// 3. VALIDAÇÃO DE RANGES (SEM RETURN)
// ═══════════════════════════════════════════════════════════════
// validação de tensões
IF (Ua < PerVar.VMIN) OR (Ua > PerVar.VMAX) THEN
    bRangeError := TRUE;
    diagnosticCode := 16#A101;  				// Erro de tensão fase A
END_IF
IF (Ub < PerVar.VMIN) OR (Ub > PerVar.VMAX) THEN
    bRangeError := TRUE;
    diagnosticCode := 16#A102;  				// Erro de tensão fase B
END_IF
IF (Uc < PerVar.VMIN) OR (Uc > PerVar.VMAX) THEN
    bRangeError := TRUE;
    diagnosticCode := 16#A103;  				// Erro de tensão fase B
END_IF

// validação de correntes
IF (ABS(Ia) > PerVar.IMAX) THEN
    bRangeError := TRUE;
    diagnosticCode := 16#A201;  				// Erro de corrente fase A
END_IF
IF (ABS(Ib) > PerVar.IMAX) THEN
    bRangeError := TRUE;
    diagnosticCode := 16#A202;  				// Erro de corrente fase B
END_IF
IF (ABS(Ic) > PerVar.IMAX) THEN
    bRangeError := TRUE;
    diagnosticCode := 16#A203;  				// Erro de corrente fase C
END_IF

// validação de potencias ativas
IF (ABS(Pt) > PerVar.PMAX) THEN
    bRangeError := TRUE;
    diagnosticCode := 16#A301;  				// Erro de potência total
END_IF
IF (ABS(Pa) > PerVar.PMAX) THEN
    bRangeError := TRUE;
    diagnosticCode := 16#A302;  				// Erro de potência Pa
END_IF
IF (ABS(Pb) > PerVar.PMAX) THEN
    bRangeError := TRUE;
    diagnosticCode := 16#A303;  				// Erro de potência Pb
END_IF
IF (ABS(Pc) > PerVar.PMAX) THEN
    bRangeError := TRUE;
    diagnosticCode := 16#A304;    				// Erro de potência Pc
END_IF

// validação de potencias reativas
IF (ABS(Qt) > PerVar.QMAX) THEN
    bRangeError := TRUE;
    diagnosticCode := 16#A401;  				// Erro de potência Qt
END_IF
IF (ABS(Qa) > PerVar.QMAX) THEN
    bRangeError := TRUE;
    diagnosticCode := 16#A402;  				// Erro de potência Qa
END_IF
IF (ABS(Qb) > PerVar.QMAX) THEN
    bRangeError := TRUE;
    diagnosticCode := 16#A403;  				// Erro de potência Qb
END_IF
IF (ABS(Qc) > PerVar.QMAX) THEN
    bRangeError := TRUE;
    diagnosticCode := 16#A404;  				// Erro de potência Qc
END_IF
	
// validação do fator das potencias
	
IF (ABS(PFt) < PFMIN) OR (ABS(PFt) >PFMAX)  THEN
    bRangeError := TRUE;
    diagnosticCode := 16#A501;  				// Erro de PFt
END_IF
IF (ABS(PFa) < PFMIN) OR (ABS(PFa) >PFMAX)  THEN
    bRangeError := TRUE;
    diagnosticCode := 16#A502;  				// Erro de PFa
END_IF
IF (ABS(PFb) < PFMIN) OR (ABS(PFb) >PFMAX)  THEN
    bRangeError := TRUE;
    diagnosticCode := 16#A503;  				// Erro de PFb
END_IF
IF (ABS(PFc) < PFMIN) OR (ABS(PFc) >PFMAX)  THEN
    bRangeError := TRUE;
    diagnosticCode := 16#A504;  				// Erro de PFc
END_IF

// ═══════════════════════════════════════════════════════════════
// 4. VALIDAÇÃO CRUZADA (SÓ SE NÃO HOUVER ERRO AINDA)
// ═══════════════════════════════════════════════════════════════

IF NOT bRangeError THEN
	// Só valida se Pa significativo (ex: > 1 kW)
	IF ABS(Pa) > 1.0 THEN
		Calculado := Ua * Ia * PFa / 1000;
		IF ABS(Pa - Calculado) > (ABS(Pa) * Tolerancia) THEN  // ✅ Usa Pa, não Calculado
			bRangeError := TRUE;
			diagnosticCode := 16#A601;
		END_IF
	END_IF
	
	// Repetir para Pb e Pc
	IF ABS(Pb) > 1.0 THEN
		Calculado := Ub * Ib * PFb / 1000;
		IF ABS(Pb - Calculado) > (ABS(Pb) * Tolerancia) THEN
			bRangeError := TRUE;
			diagnosticCode := 16#A602;
		END_IF
	END_IF
	
	IF ABS(Pc) > 1.0 THEN
		Calculado := Uc * Ic * PFc / 1000;
		IF ABS(Pc - Calculado) > (ABS(Pc) * Tolerancia) THEN
			bRangeError := TRUE;
			diagnosticCode := 16#A603;
		END_IF
	END_IF
	// Pt = Pa + Pb + Pc
	SomaP := Pa + Pb + Pc;
	IF ABS(Pt) > 1.0 THEN  // ✅ Só valida se significativo
		IF ABS(Pt - SomaP) > (ABS(Pt) * Tolerancia) THEN  // ✅ Usa Pt
			bRangeError := TRUE;
			diagnosticCode := 16#A604;
		END_IF
	END_IF
	
	// FPt com base nas potencias ativas e reativas
	SomaQ:=Qa + Qb + Qc;
	Calculado := SQRT((SomaP * SomaP)+ (SomaQ * SomaQ));
	IF Calculado > 10 THEN 									// 1 kva
		Calculado := SomaP / Calculado;
		IF ABS(PFt - Calculado) > 0.05 THEN
			bRangeError := TRUE;
			diagnosticCode := 16#A605;  
		END_IF
	END_IF
END_IF;

// ═══════════════════════════════════════════════════════════════
// 5. DETECÇÃO DE CONGELAMENTO (OPCIONAL)
// ═══════════════════════════════════════════════════════════════
IF NOT bRangeError THEN
	IF ABS(Pt - Pt_last) < 1.0 THEN  // < 1 kW de variação
		frozen_count := frozen_count + 1;
	ELSE
		frozen_count := 0;
	END_IF
	
	IF frozen_count > FREEZE_THRESHOLD THEN
		bRangeError := TRUE;
		diagnosticCode := 16#A900;
	END_IF
END_IF

Pt_last := Pt;
// ═══════════════════════════════════════════════════════════════
// 6. TRATAMENTO FINAL DE ERRO/SUCESSO
// ═══════════════════════════════════════════════════════==══════
IF bRangeError THEN
	
    nErrors := MIN(nErrors + 1, 10);  // Clamp em 10
    bDadosOK := FALSE;  // Dado atual é inválido
    
    IF nErrors >= 5 THEN
        bPoucosErros := FALSE;  // 🚨 Degradação crítica
    ELSE
        bPoucosErros := TRUE;   // ⚠️ Ainda tolerável (1-4 erros)
    END_IF
    // ❌ NÃO atualiza variáveis globais (mantém último valor válido)
    // ❌ NÃO reseta filtro (preserva estado anterior)  
ELSE
	// 1. Decrementa contador de erros (recuperação gradual)
    IF nErrors > 0 THEN
        nErrors := nErrors - 1;
    END_IF
    
    bDadosOK := TRUE;
    bPoucosErros := TRUE;
    diagnosticCode := 0;
	
    // 2. FILTRO PASSA-BAIXA (Suavização de Medição)
    // ─────────────────────────────────────────────────────────
    IF bFirstRun THEN
        Pt_filt := Pt;
        Qt_filt := Qt;
        PFt_filt := PFt;
        bFirstRun := FALSE;
    ELSE
		// Filtro exponencial: y[n] = α·x[n] + (1-α)·y[n-1]
        // ALPHA configurável (ex: 0.25 → ~3s para 95% do valor)
        Pt_filt := PerVar.ALPHA * Pt + (1.0 - PerVar.ALPHA) * Pt_filt;
        Qt_filt := PerVar.ALPHA * Qt + (1.0 - PerVar.ALPHA) * Qt_filt;
        PFt_filt := PerVar.ALPHA * PFt + (1.0 - PerVar.ALPHA) * PFt_filt;
    END_IF
	
	// 3. ATUALIZAÇÃO DE VARIÁVEIS GLOBAIS
    // ──────────────────────────────────────────────────────────
	Global.Ua  := Ua;				// em Volts
	Global.Ub  := Ub;				// em Volts
	Global.Uc  := Uc;				// em Volts
	
	Global.Ia  := Ia;				// em Amperes
	Global.Ib  := Ib;				// em Amperes
	Global.Ic  := Ic;				// em Amperes
	
	// Potência Ativa (FILTRADA para controle)
	Global.Pt  := Pt_filt;			// kW
	Global.Pa  := Pa;				// kW
	Global.Pb  := Pb;				// kW
	Global.Pc  := Pc;				// kW
	
	// Potência Reativa (FILTRADA para controle de PF)
	Global.Qt  := Qt_filt;			// kvar
	Global.Qa  := Qa;				// kvar
	Global.Qb  := Qb;				// kvar
	Global.Qc  := Qc;				// kvar
    
    // Fator de Potência (FILTRADO para controle)
	Global.PFt := PFt_filt;				
	Global.PFa := PFa;
	Global.PFb := PFb;
	Global.PFc := PFc;

END_IF

END_FUNCTION_BLOCK

// Dispositivo/Application/FB_WriteInv
FUNCTION_BLOCK FB_WriteInv

VAR_INPUT
    Execute     : BOOL;
    InvIndex    : UINT;
END_VAR

VAR_IN_OUT
    trigInv     : BOOL;                    // ex.: Global.trigInvCOM100[i]
    pSlave      : ModbusSlaveComPort;      // ex.: Global.pInversores100[i]^
END_VAR

VAR_OUTPUT
    result      : E_ModbusResult;
END_VAR

VAR
    fbAlarmes   : FB_Alarmes;
    fbChannel   : ModbusChannel;
    state       : (TRIG, WAIT) := TRIG;
    tonTimer    : TON;
    tTimeout    : TIME := T#150MS;
END_VAR

// ============================================================
// Máquina de estados de escrita em inversores
// ============================================================

// estado default por ciclo
result := E_ModbusResult.BUSY;

// bloqueio por Execute
IF NOT Execute THEN
    trigInv := FALSE;
    state := TRIG;
    result := E_ModbusResult.END;
    RETURN;
END_IF

tonTimer(IN := (state = WAIT), PT := tTimeout);

CASE state OF

    TRIG:
        trigInv := TRUE;
        state := WAIT;

    WAIT:
       IF pSlave.xDone THEN
            trigInv := FALSE;
            state := TRIG;
            result := E_ModbusResult.DONE;
			
		
      	ELSIF pSlave.xError THEN
            fbChannel(Slave := pSlave, iChannelIndex := 0);
            fbAlarmes(codigo := fbChannel.ModbusError,tError := TO_UDINT(SysTimeRtcGet(Global.Result)));
            state := TRIG;
            trigInv := FALSE;
            result := E_ModbusResult.ERRO;
			
      	ELSIF tonTimer.Q THEN
            fbAlarmes(codigo := 16#B2,tError := TO_UDINT(SysTimeRtcGet(Global.Result)));
            state := TRIG;
            trigInv := FALSE;
            result := E_ModbusResult.TIMEOUT;
        END_IF
END_CASE

END_FUNCTION_BLOCK

// Dispositivo/Application/FB_ValidaDadosMedidor
(*═════════════════════════════════════════════════════════════════════
 FB_ValidaMedicao
 
 Valida medições do medidor trifásico via Modbus, aplica filtro
 passa-baixa e verifica consistência física das grandezas.
 
 ENTRADAS:
 - (nenhuma - lê de valorLido.WordArray via Modbus)
 
 SAÍDAS:
 - bDadosOK: TRUE se medições são válidas
 - bPoucosErros: TRUE se < 5 erros consecutivos
 - diagnosticCode: Código de falha (0 = OK)
 
 LÓGICA:
 1. Conversão de escalas (Modbus → unidades físicas)
 2. Validação de ranges individuais
 3. Validação cruzada (Pt vs soma, PF vs P/S)
 4. Detecção de congelamento 
 5. Filtro passa-baixa exponencial (SOMENTE se validação OK)
 6. Atualização de variáveis globais (SOMENTE se validação OK)
 7. Janela de erros (5 consecutivos = FAIL_SAFE)
═════════════════════════════════════════════════════════════════════*)
FUNCTION_BLOCK FB_ValidaDadosMedidor

VAR_OUTPUT
    bDadosOK		: BOOL 	:= FALSE;  // Dados aprovados
	bPoucosErros	: BOOL  := TRUE;  // Inicialmente sem erros
    diagnosticCode 	: WORD;            // Código de falha
END_VAR

VAR
	valorLido		: UN_Rele;
	Ua    	    	: REAL := 0.0; // 2006H - Tensão de fase A x 0,1 V
	Ub    	    	: REAL := 0.0; // 2008H - Tensão de fase B x 0,1 V
	Uc    	    	: REAL := 0.0; // 200AH - Tensão de fase C x 0,1 V
	
	Ia    	    	: REAL := 0.0; // 200CH - Corrente de fase A x 0,001 A 
	Ib    	    	: REAL := 0.0; // 200EH - Corrente de fase B x 0,001 A
	Ic    	    	: REAL := 0.0; // 2010H - Corrente de fase C x 0,001 A
	
	Pt    	    	: REAL := 0.0; // 2012H - Potencia ativa combinada x 0,1 W
	Pa    	    	: REAL := 0.0; // 2014H - Potencia ativa fase A x 0,1 W
	Pb    	    	: REAL := 0.0; // 2016H - Potencia ativa fase B x 0,1 W
	Pc    	   		: REAL := 0.0; // 2018H - Potencia ativa fase C x 0,1 W	
		
	Qt    	    	: REAL := 0.0; // 201AH - Potencia reativa combinada x 0,1 var
	Qa    	    	: REAL := 0.0; // 201CH - Potencia reativa fase A x 0,1 var
	Qb    	    	: REAL := 0.0; // 201EH - Potencia reativa fase B x 0,1 var
	Qc    	    	: REAL := 0.0; // 2020H - Potencia reativa fase C x 0,1 var

	PFt    	    	: REAL := 0.0; // 202AH - Fator de potência combinado (número positivo: indutivo, número negativo: capacitivo) (x  0,001)
	PFa    	    	: REAL := 0.0; // 202CH - Fator de potência de fase A (número positivo: indutivo, número negativo: capacitivo)  (×0,001)
	PFb    	    	: REAL := 0.0; // 202EH - Fator de potência de fase B (número positivo: indutivo, número negativo: capacitivo)  (×0,001)
	PFc    	    	: REAL := 0.0; // 2030H - Fator de potência de fase C (número positivo: indutivo, número negativo: capacitivo)  (×0,001)
	
	// Limites físicos (ajustar conforme instalação)
    PFMIN 			: REAL := 0.5;
    PFMAX 			: REAL := 1.0;
	
	// variaveis auxiliares
    bRangeError 	: BOOL := FALSE;            // Fora de faixa
	nErrors 		: UINT := 0;
	SomaP			: REAL;
	SomaQ 			: REAL;
	Calculado 		: REAL;
	Tolerancia  	: REAL :=0.05;
	Pt_last 		: REAL := 0.0;
    frozen_count 	: UINT := 0;
	FREEZE_THRESHOLD: UINT := 10;  		// 10 ciclos
	bFirstRun		: BOOL :=TRUE;
	Pt_filt 		: REAL :=0;
    Qt_filt 		: REAL :=0;
    PFt_filt 		: REAL :=0;
END_VAR

// ═══════════════════════════════════════════════════════════════
// 1. RESET DE ESTADO
// ═══════════════════════════════════════════════════════════════

bRangeError := FALSE;
diagnosticCode := 0;

// ═══════════════════════════════════════════════════════════════
// 2. CONVERSÃO DE ESCALAS
// ═══════════════════════════════════════════════════════════════
Ua  := valorLido.EmReal.Ua * 0.1;				// em Volts
Ub  := valorLido.EmReal.Ub * 0.1;				// em Volts
Uc  := valorLido.EmReal.Uc * 0.1;				// em Volts

Ia  := valorLido.EmReal.Ia * 0.001;				// em Amperes
Ib  := valorLido.EmReal.Ib * 0.001;				// em Amperes
Ic  := valorLido.EmReal.Ic * 0.001;				// em Amperes

Pt  := valorLido.EmReal.Pt *0.0001;				// kW
Pa  := valorLido.EmReal.Pa *0.0001;				// kW
Pb  := valorLido.EmReal.Pb *0.0001;				// kW
Pc  := valorLido.EmReal.Pc *0.0001;				// kW

Qt  := valorLido.EmReal.Qt *0.0001;				// kvar
Qa  := valorLido.EmReal.Qa *0.0001;				// kvar
Qb  := valorLido.EmReal.Qb *0.0001;				// kvar
Qc  := valorLido.EmReal.Qc *0.0001;				// xkvar

PFt := valorLido.EmReal.PFt *0.001;	
PFa := valorLido.EmReal.PFa *0.001;
PFb := valorLido.EmReal.PFb *0.001;
PFc := valorLido.EmReal.PFc *0.001;

// ═══════════════════════════════════════════════════════════════
// 3. VALIDAÇÃO DE RANGES (SEM RETURN)
// ═══════════════════════════════════════════════════════════════
// validação de tensões
IF (Ua < PerVar.VMIN) OR (Ua > PerVar.VMAX) THEN
    bRangeError := TRUE;
    diagnosticCode := 16#A101;  				// Erro de tensão fase A
END_IF
IF (Ub < PerVar.VMIN) OR (Ub > PerVar.VMAX) THEN
    bRangeError := TRUE;
    diagnosticCode := 16#A102;  				// Erro de tensão fase B
END_IF
IF (Uc < PerVar.VMIN) OR (Uc > PerVar.VMAX) THEN
    bRangeError := TRUE;
    diagnosticCode := 16#A103;  				// Erro de tensão fase B
END_IF

// validação de correntes
IF (ABS(Ia) > PerVar.IMAX) THEN
    bRangeError := TRUE;
    diagnosticCode := 16#A201;  				// Erro de corrente fase A
END_IF
IF (ABS(Ib) > PerVar.IMAX) THEN
    bRangeError := TRUE;
    diagnosticCode := 16#A202;  				// Erro de corrente fase B
END_IF
IF (ABS(Ic) > PerVar.IMAX) THEN
    bRangeError := TRUE;
    diagnosticCode := 16#A203;  				// Erro de corrente fase C
END_IF

// validação de potencias ativas
IF (ABS(Pt) > PerVar.PMAX) THEN
    bRangeError := TRUE;
    diagnosticCode := 16#A301;  				// Erro de potência total
END_IF
IF (ABS(Pa) > PerVar.PMAX) THEN
    bRangeError := TRUE;
    diagnosticCode := 16#A302;  				// Erro de potência Pa
END_IF
IF (ABS(Pb) > PerVar.PMAX) THEN
    bRangeError := TRUE;
    diagnosticCode := 16#A303;  				// Erro de potência Pb
END_IF
IF (ABS(Pc) > PerVar.PMAX) THEN
    bRangeError := TRUE;
    diagnosticCode := 16#A304;    				// Erro de potência Pc
END_IF

// validação de potencias reativas
IF (ABS(Qt) > PerVar.QMAX) THEN
    bRangeError := TRUE;
    diagnosticCode := 16#A401;  				// Erro de potência Qt
END_IF
IF (ABS(Qa) > PerVar.QMAX) THEN
    bRangeError := TRUE;
    diagnosticCode := 16#A402;  				// Erro de potência Qa
END_IF
IF (ABS(Qb) > PerVar.QMAX) THEN
    bRangeError := TRUE;
    diagnosticCode := 16#A403;  				// Erro de potência Qb
END_IF
IF (ABS(Qc) > PerVar.QMAX) THEN
    bRangeError := TRUE;
    diagnosticCode := 16#A404;  				// Erro de potência Qc
END_IF
	
// validação do fator das potencias
	
IF (ABS(PFt) < PFMIN) OR (ABS(PFt) >PFMAX)  THEN
    bRangeError := TRUE;
    diagnosticCode := 16#A501;  				// Erro de PFt
END_IF
IF (ABS(PFa) < PFMIN) OR (ABS(PFa) >PFMAX)  THEN
    bRangeError := TRUE;
    diagnosticCode := 16#A502;  				// Erro de PFa
END_IF
IF (ABS(PFb) < PFMIN) OR (ABS(PFb) >PFMAX)  THEN
    bRangeError := TRUE;
    diagnosticCode := 16#A503;  				// Erro de PFb
END_IF
IF (ABS(PFc) < PFMIN) OR (ABS(PFc) >PFMAX)  THEN
    bRangeError := TRUE;
    diagnosticCode := 16#A504;  				// Erro de PFc
END_IF

// ═══════════════════════════════════════════════════════════════
// 4. VALIDAÇÃO CRUZADA (SÓ SE NÃO HOUVER ERRO AINDA)
// ═══════════════════════════════════════════════════════════════

IF NOT bRangeError THEN
	// Só valida se Pa significativo (ex: > 1 kW)
	IF ABS(Pa) > 1.0 THEN
		Calculado := Ua * Ia * PFa / 1000;
		IF ABS(Pa - Calculado) > (ABS(Pa) * Tolerancia) THEN  // ✅ Usa Pa, não Calculado
			bRangeError := TRUE;
			diagnosticCode := 16#A601;
		END_IF
	END_IF
	
	// Repetir para Pb e Pc
	IF ABS(Pb) > 1.0 THEN
		Calculado := Ub * Ib * PFb / 1000;
		IF ABS(Pb - Calculado) > (ABS(Pb) * Tolerancia) THEN
			bRangeError := TRUE;
			diagnosticCode := 16#A602;
		END_IF
	END_IF
	
	IF ABS(Pc) > 1.0 THEN
		Calculado := Uc * Ic * PFc / 1000;
		IF ABS(Pc - Calculado) > (ABS(Pc) * Tolerancia) THEN
			bRangeError := TRUE;
			diagnosticCode := 16#A603;
		END_IF
	END_IF
	// Pt = Pa + Pb + Pc
	SomaP := Pa + Pb + Pc;
	IF ABS(Pt) > 1.0 THEN  // ✅ Só valida se significativo
		IF ABS(Pt - SomaP) > (ABS(Pt) * Tolerancia) THEN  // ✅ Usa Pt
			bRangeError := TRUE;
			diagnosticCode := 16#A604;
		END_IF
	END_IF
	
	// FPt com base nas potencias ativas e reativas
	SomaQ:=Qa + Qb + Qc;
	Calculado := SQRT((SomaP * SomaP)+ (SomaQ * SomaQ));
	IF Calculado > 10 THEN 									// 1 kva
		Calculado := SomaP / Calculado;
		IF ABS(PFt - Calculado) > 0.05 THEN
			bRangeError := TRUE;
			diagnosticCode := 16#A605;  
		END_IF
	END_IF
END_IF;

// ═══════════════════════════════════════════════════════════════
// 5. DETECÇÃO DE CONGELAMENTO (OPCIONAL)
// ═══════════════════════════════════════════════════════════════
IF NOT bRangeError THEN
	IF ABS(Pt - Pt_last) < 1.0 THEN  // < 1 kW de variação
		frozen_count := frozen_count + 1;
	ELSE
		frozen_count := 0;
	END_IF
	
	IF frozen_count > FREEZE_THRESHOLD THEN
		bRangeError := TRUE;
		diagnosticCode := 16#A900;
	END_IF
END_IF

Pt_last := Pt;
// ═══════════════════════════════════════════════════════════════
// 6. TRATAMENTO FINAL DE ERRO/SUCESSO
// ═══════════════════════════════════════════════════════==══════
IF bRangeError THEN
	
    nErrors := MIN(nErrors + 1, 10);  // Clamp em 10
    bDadosOK := FALSE;  // Dado atual é inválido
    
    IF nErrors >= 5 THEN
        bPoucosErros := FALSE;  // 🚨 Degradação crítica
    ELSE
        bPoucosErros := TRUE;   // ⚠️ Ainda tolerável (1-4 erros)
    END_IF    
    // ❌ NÃO atualiza variáveis globais (mantém último valor válido)
    // ❌ NÃO reseta filtro (preserva estado anterior)  
ELSE
	// 1. Decrementa contador de erros (recuperação gradual)
    IF nErrors > 0 THEN
        nErrors := nErrors - 1;
    END_IF
    
    bDadosOK := TRUE;
    bPoucosErros := TRUE;
    diagnosticCode := 0;
	
    // 2. FILTRO PASSA-BAIXA (Suavização de Medição)
    // ─────────────────────────────────────────────────────────
    IF bFirstRun THEN
        Pt_filt := Pt;
        Qt_filt := Qt;
        PFt_filt := PFt;
        bFirstRun := FALSE;
    ELSE
		// Filtro exponencial: y[n] = α·x[n] + (1-α)·y[n-1]
        // ALPHA configurável (ex: 0.25 → ~3s para 95% do valor)
        Pt_filt := PerVar.ALPHA * Pt + (1.0 - PerVar.ALPHA) * Pt_filt;
        Qt_filt := PerVar.ALPHA * Qt + (1.0 - PerVar.ALPHA) * Qt_filt;
        PFt_filt := PerVar.ALPHA * PFt + (1.0 - PerVar.ALPHA) * PFt_filt;
    END_IF
	
	// 3. ATUALIZAÇÃO DE VARIÁVEIS GLOBAIS
    // ──────────────────────────────────────────────────────────
	Global.Ua  := Ua;				// em Volts
	Global.Ub  := Ub;				// em Volts
	Global.Uc  := Uc;				// em Volts
	
	Global.Ia  := Ia;				// em Amperes
	Global.Ib  := Ib;				// em Amperes
	Global.Ic  := Ic;				// em Amperes
	
	// Potência Ativa (FILTRADA para controle)
	Global.Pt  := Pt_filt;			// kW
	Global.Pa  := Pa;				// kW
	Global.Pb  := Pb;				// kW
	Global.Pc  := Pc;				// kW
	
	// Potência Reativa (FILTRADA para controle de PF)
	Global.Qt  := Qt_filt;			// kvar
	Global.Qa  := Qa;				// kvar
	Global.Qb  := Qb;				// kvar
	Global.Qc  := Qc;				// kvar
    
    // Fator de Potência (FILTRADO para controle)
	Global.PFt := PFt_filt;				
	Global.PFa := PFa;
	Global.PFb := PFb;
	Global.PFc := PFc;

END_IF

END_FUNCTION_BLOCK

// Dispositivo/Application/Pages/Alarms
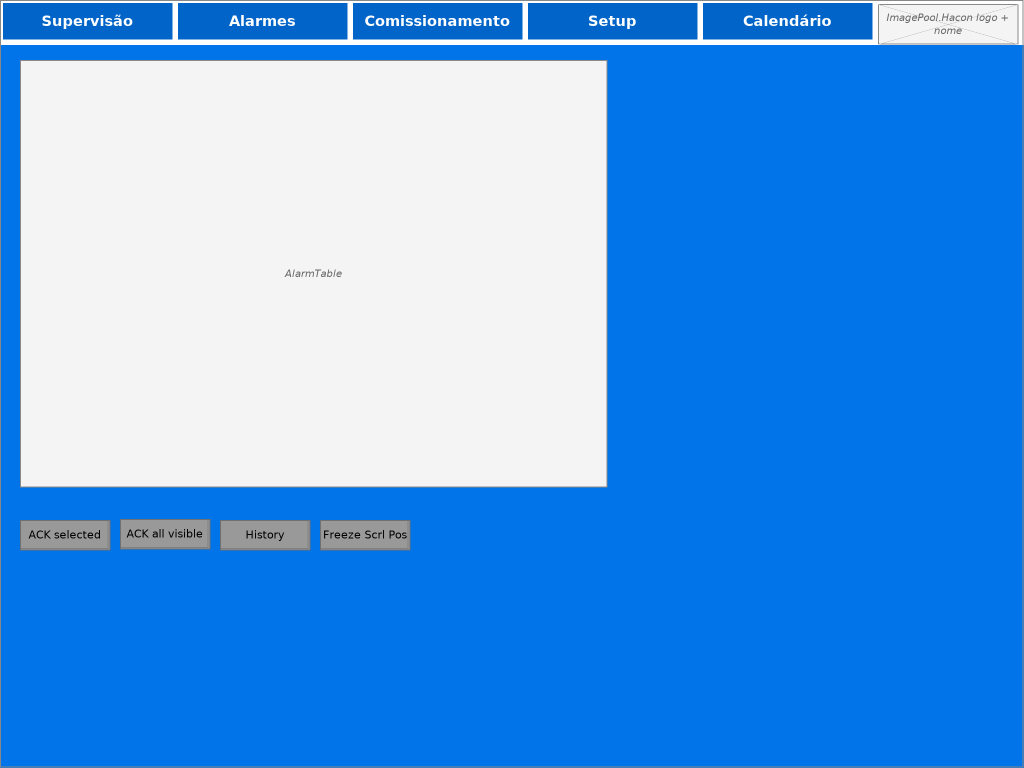
VISUALIZATION Alarms  // 1024x768
VAR_IN_OUT
END_VAR
VAR
	bAckSel : BOOL;
	bAckVisible : BOOL;
	bHistory : BOOL;
	bFreezeScrlPos : BOOL;
END_VAR
    Frame (0,0 1024x768)
        shows Template()
    AlarmTable (20,60 587x427)
        p1521930926: __All
        p1663851261: __All
        p428520879: bAckSel
        p2607059081: bAckVisible
        p3266827225: bHistory
        p3894972949: bFreezeScrlPos
    Button (20,520 90x30), "ACK selected"
        toggle bAckSel
    Button (120,519 90x30), "ACK all visible"
        toggle bAckVisible
    Button (220,520 90x30), "History"
        toggle bHistory
    Button (320,520 90x30), "Freeze Scrl Pos"
        toggle bFreezeScrlPos
END_VISUALIZATION

